{attribute 'GeneratedUsingTerminal: EL6001-0000-0020'}
{attribute addProperty BoxType "EL6001-0000-0020"}
{attribute addProperty Id "CtrlAT %Q*USINT1Data_OutAT %Q*ARRAY[0..4] OF USINT5"}
{attribute addProperty CRC "799778629"}
{attribute addProperty Size "6"}
TYPE Outputs_2CF06B6A :
STRUCT
	{attribute addProperty Name "Ctrl"}
	Ctrl AT %Q* : USINT;
	{attribute addProperty Name "Data_Out"}
	Data_Out AT %Q* : ARRAY[0..4] OF USINT;
END_STRUCT
END_TYPE

(* stored: Version 1.2.0.0, ProductVersion 3.1.4024.9
   DUT Outputs_2CF06B6A: Id {416097cc-b585-4be9-90ca-8b1f9da61b99} *)
